SUBAPPLICATION Uebung_039a_sub_Outputs (* Subapplication Type *)
  (* Standard: 61499-2 *)
  (* Version 1.0, 2024-03-03, franz *)
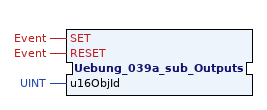
  EVENT_INPUT
    SET; (* Set Output *)
    RESET; (* Reset Output *)
  END_EVENT
  VAR_INPUT
    u16ObjId : UINT := ID_NULL; (* Object ID Softkey/Button *)
  END_VAR
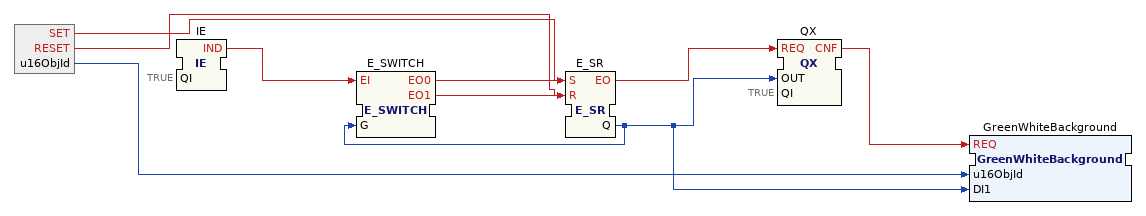
  FBS
    QX : QX(QI := TRUE);
    E_SWITCH : E_SWITCH;
    E_SR : E_SR;
    IE : IE(QI := TRUE);
  END_FBS
  SUBAPPS
    GreenWhiteBackground : GreenWhiteBackground;
  END_SUBAPPS
  EVENT_CONNECTIONS
    QX.CNF TO GreenWhiteBackground.REQ;
    E_SWITCH.EO0 TO E_SR.S;
    E_SWITCH.EO1 TO E_SR.R;
    IE.IND TO E_SWITCH.EI;
    E_SR.EO TO QX.REQ;
    SET TO E_SR.S;
    RESET TO E_SR.R;
  END_CONNECTIONS
  DATA_CONNECTIONS
    u16ObjId TO GreenWhiteBackground.u16ObjId;
    E_SR.Q TO E_SWITCH.G;
    E_SR.Q TO QX.OUT;
    E_SR.Q TO GreenWhiteBackground.DI1;
  END_CONNECTIONS
END_SUBAPPLICATION
